{attribute addProperty BoxType "EL2878-0005-0016"}
{attribute addProperty Id "DiagAT %I*BOOL81"}
{attribute addProperty CRC "1289020322"}
{attribute addProperty SizeInBites "8"}
{attribute addProperty SizeInBytes "1"}
TYPE Diagnostic_4CD4E3A2 :
STRUCT
	{attribute addProperty Name "Diag"}
	Diag AT %I* : BOOL;
END_STRUCT
END_TYPE

(* stored: Version 1.2.0.0, ProductVersion 3.1.4024.9
   DUT Diagnostic_4CD4E3A2: Id {28d5d3a1-8a71-430a-9e71-87d631408358} *)
